// TIA Portal project "Práctica 10 potencia" (V15)

(* hardware
DEVICE "S7-1200 station_1"  S7-1200 Station
   slot 0: "Rack_0"  S7-1200 Rack  Rack  V1.0
   slot 1: "PLC_1"  CPU 1214C AC/DC/Rly  6ES7 214-1BG40-0XB0  V4.2
   slot 3: "AQ 1x12BIT_1"  AQ1 signal board  6ES7 232-4HA30-0XB0  V1.0
DEVICE "HMI_1"  KTP700 Basic PN
   slot 0: "HMI_1"  KTP700 Basic PN  6AV2 123-2GB03-0AX0  15.0.0.0
   slot 1: "HMI_RT_1"  KTP700 Basic PN  6AV2 123-2GB03-0AX0  15.0.0.0
   slot 5: "HMI_1.IE_CP_1"  PROFINET Interface  15.0.0.0
      slot 1: "Interfaz PROFINET_1"  PROFINET Interface
         slot 1: "Port_1"  Port
*)

// ===== PLC "PLC_1"  CPU 1214C AC/DC/Rly =====

VAR_GLOBAL   // PLC tag table "Tabla de variables estándar"
   "S" AT %MD30 : Real;
   "Q" AT %MD34 : Real;
   "P" AT %MD38 : Real;
   "FDP" AT %MD42 : Real;
   "Sumado" AT %MD46 : Real;
   "P2" AT %MD50 : Real;
   "Calcular" AT %M5.1 : Bool;
   "Q2" AT %MD54 : Real;
   "FDP2" AT %MD58 : Real;
   "FI" AT %MD62 : Real;
   "ANGULO" AT %MD66 : Real;
   "ALFA" AT %MD70 : Real;
   "Tag_1" AT %MD80 : Real;
   "P Y Q DIV" AT %MD84 : Real;
END_VAR

FUNCTION "angulos" : Void   // FC1, LAD
{ S7_Optimized_Access := 'TRUE' }
VERSION : 0.1
   VAR_INPUT
      deg_i : Real;
      rad_i : Real;
   END_VAR
   VAR_OUTPUT
      deg_o : Real;
      rad_o : Real;
   END_VAR
   VAR_TEMP
      k1 : Real;
      k2 : Real;
   END_VAR
BEGIN

REGION Network 1
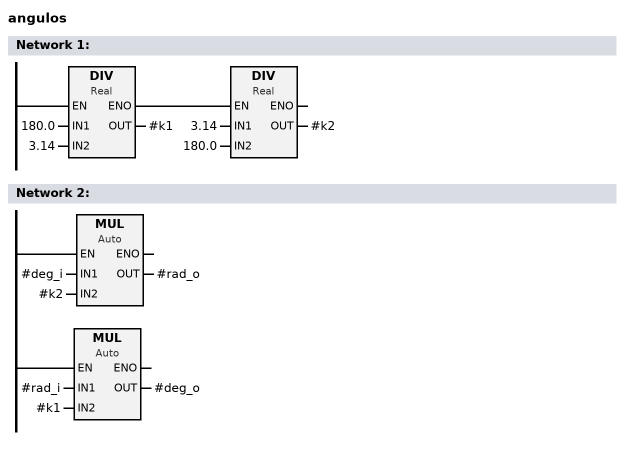
   RUNG wire#powerrail
      { S7_Templates := "SrcType := Real" } Div(in1 := 180.0, in2 := 3.14, out => #k1)
      { S7_Templates := "SrcType := Real" } Div(in1 := 3.14, in2 := 180.0, out => #k2)
   END_RUNG
   // the same network as SCL:
   #k1 := 180.0 / 3.14;
   #k2 := 3.14 / 180.0;
END_REGION

REGION Network 2
   RUNG wire#powerrail
      Mul(in1 := #deg_i, in2 := #k2, out => #rad_o)
   END_RUNG
   RUNG wire#powerrail
      Mul(in1 := #rad_i, in2 := #k1, out => #deg_o)
   END_RUNG
   // the same network as SCL:
   #rad_o := #deg_i * #k2;
   #deg_o := #rad_i * #k1;
END_REGION
END_FUNCTION

FUNCTION "pitágoras" : Void   // FC2, LAD
{ S7_Optimized_Access := 'TRUE' }
VERSION : 0.1
   VAR_INPUT
      P : Real;
      Q : Real;
   END_VAR
   VAR_OUTPUT
      S : Real;
      FDP_1 : Real;
   END_VAR
   VAR_TEMP
      P2 : Real;
      Q2 : Real;
      Sumado : Real;
      FDP : Real;
   END_VAR
BEGIN

REGION Network 1: Pitágoras
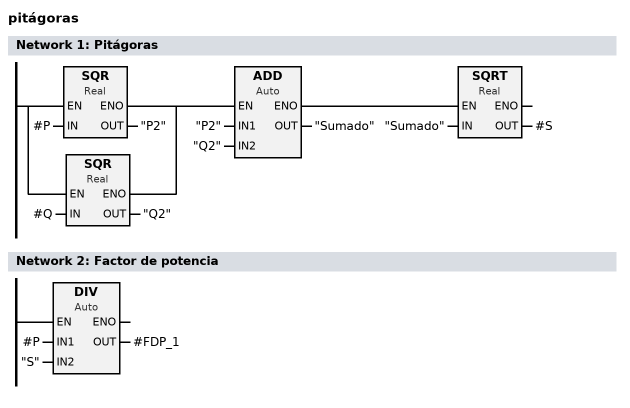
   "P2" := SQR(#P);
   "Q2" := SQR(#Q);
   IF TRUE OR TRUE THEN
       "Sumado" := "P2" + "Q2";
       #S := SQRT("Sumado");
   END_IF;
END_REGION

REGION Network 2: Factor de potencia
   RUNG wire#powerrail
      Div(in1 := #P, in2 := "S", out => #FDP_1)
   END_RUNG
   // the same network as SCL:
   #FDP_1 := #P / "S";
END_REGION
END_FUNCTION

ORGANIZATION_BLOCK "Main"   // OB1, LAD, ProgramCycle
TITLE = "Main Program Sweep (Cycle)"
{ S7_Optimized_Access := 'TRUE' }
VERSION : 0.1
   VAR_INPUT
      Initial_Call : Bool;   // Initial call of this OB
      Remanence : Bool;   // =True, if remanent data are available
   END_VAR
BEGIN

REGION Network 1: Operación para sacar FDP
   // Sabiendo dos lados del triángulo, con la función "pitagoras" sacamos la hipotenusa y el factor de potencia.
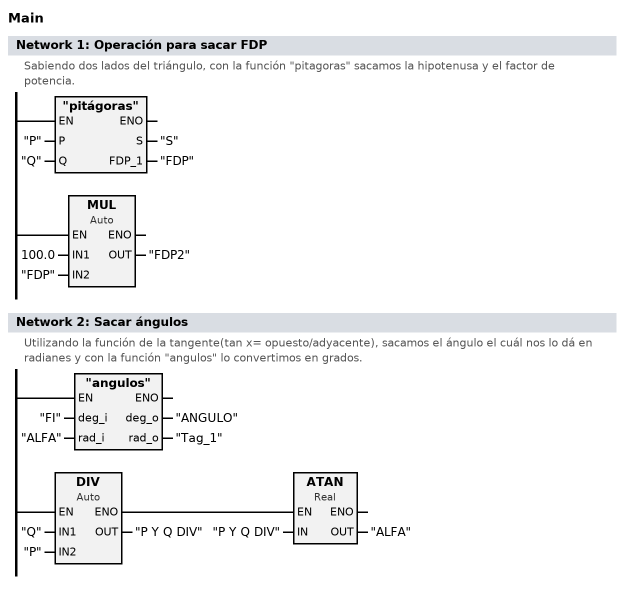
   RUNG wire#powerrail
      "pitágoras"(P := "P", Q := "Q", S => "S", FDP_1 => "FDP")
   END_RUNG
   RUNG wire#powerrail
      Mul(in1 := 100.0, in2 := "FDP", out => "FDP2")
   END_RUNG
   // the same network as SCL:
   "pitágoras"(P := "P", Q := "Q", S => "S", FDP_1 => "FDP");
   "FDP2" := 100.0 * "FDP";
END_REGION

REGION Network 2: Sacar ángulos
   // Utilizando la función de la tangente(tan x= opuesto/adyacente), sacamos el ángulo el cuál nos lo dá en radianes y con la función "angulos" lo convertimos en grados.
   "angulos"(deg_i := "FI", rad_i := "ALFA", deg_o => "ANGULO", rad_o => "Tag_1");
   "P Y Q DIV" := "Q" / "P";
   "ALFA" := ATAN("P Y Q DIV");
END_REGION
END_ORGANIZATION_BLOCK

(* ===== HMI "HMI_RT_1" =====
system functions are stored by id; their names below are inferred from use
connection "HMI_Conexión_1": ETHERNET, SMART_S7_1200_OMS

HMI tags "Tabla de variables estándar"
   "Número_imagen_variable" : UInt, internal
   "P" : Real = PLC P AT %MD38, 1 s
   "Q" : Real = PLC Q AT %MD34, 1 s
   "S" : Real = PLC S AT %MD30, 1 s
   "Calcular" : Bool = PLC Calcular AT %M5.1, 1 s
   "FDP" : Real = PLC FDP AT %MD42, 1 s
   "FDP2" : Real = PLC FDP2 AT %MD58, 1 s
   "ANGULO" : Real = PLC ANGULO AT %MD66, 1 s

text list "Nombre_imagen_lista_texto": 1 'Imagen raíz'

Template "Plantilla_1" 800x480
   Button "Salir" at 714,429 size 71x50; TextOff 'Salir'; PictureOff "ExitRuntime_KTP700_Basic_PN_TR"; PictureOn "ExitRuntime_KTP700_Basic_PN_TR"
      on Release: StopRuntime(0)
   Button "Template_Button" at 614,429 size 71x50; TextOff 'Text'
   Button "Template_Button_1" at 514,429 size 71x50; TextOff 'Text'
   Button "Template_Button_2" at 414,429 size 71x50; TextOff 'Text'
   Button "Template_Button_3" at 314,429 size 71x50; TextOff 'Text'
   Button "Template_Button_4" at 214,429 size 71x50; TextOff 'Text'
   Button "Avisos" at 114,429 size 71x50; TextOff 'Avisos'; PictureOff "AlarmDisplay_KTP700_Basic_PN_TR"; PictureOn "AlarmDisplay_KTP700_Basic_PN_TR"
      on Release: function_ef3f5d25("Ventana de avisos_no_acusado", -1)
   Button "Imagen inicial" at 14,429 size 71x50; TextOff 'Imagen inicial'; PictureOff "NavigateHome_KTP700_Basic_PN_TR"; PictureOn "NavigateHome_KTP700_Basic_PN_TR"
      on Release: ActivateScreen("Imagen raíz", 0)
   SymbolicIOField "Imagen_campo_ES_simbólico" at 93,9 size 600x33; TextOff '0'; TextOn '1'; TextList "Nombre_imagen_lista_texto"
      ProcessValue <- "Número_imagen_variable"
      on Change: ActivateScreenByNumber("Número_imagen_variable", 0)
   DateTimeField "HmiScreenItemData" at 695,25 size 105x25
   DateTimeField "HmiScreenItemData_1" at 695,0 size 105x25
   GraphicView "Logotipo" at 0,0 size 91x51; Picture "Logotipo de HMI_1"

screen "Imagen raíz" 800x480, template "Plantilla_1"
   on GenerateScreen: SetTag("Número_imagen_variable", 1)
   TextField "Campo de texto_1" at 242,104 size 21x34; Text 'S'
   TextField "Campo de texto_2" at 490,150 size 24x34; Text 'Q'
   TextField "Campo de texto_3" at 303,258 size 21x34; Text 'P'
   TextField "Campo de texto_4" at 258,373 size 109x34; Text 'FDP'
   IOField "Campo ES_1" at 331,258 size 107x34
      ProcessValue <- "P"
   IOField "Campo ES_2" at 519,147 size 103x34
      ProcessValue <- "Q"
   IOField "Campo ES_3" at 276,105 size 95x36
      ProcessValue <- "S"
   IOField "Campo ES_4" at 331,373 size 130x32; FormatPattern 99.999
      ProcessValue <- "FDP"
   Circle "Círculo_1" at 511,368 size 52x52
      Appearance <- "FDP2"
   IOField "Campo ES_5" at 283,210 size 96x32
      ProcessValue <- "ANGULO"
   TextField "Campo de texto_5" at 253,222 size 18x28; Text 'α'
*)